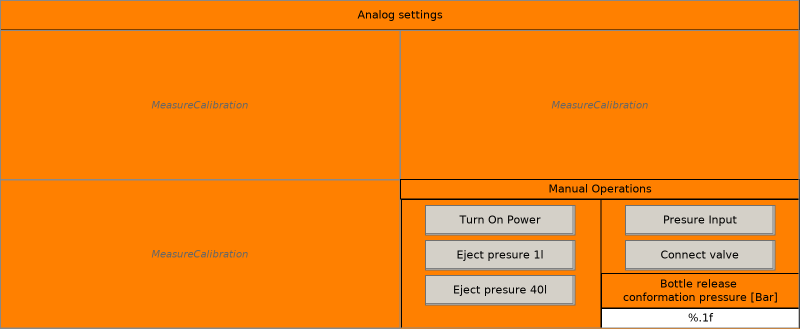
VISUALIZATION vService  // 800x329
VAR_IN_OUT
	fbChamber 	: fbChamber;
	stParams	: stParamsChamber;
END_VAR
    Rectangle (600,199 200x129)
    Rectangle (401,199 200x129)
    Rectangle (0,0 800x30), "Analog settings"
    Frame (0,30 400x150)
        shows MeasureCalibration(stMeasureData := stParams.stPressureSens, diAnalogIn := fbChamber.stInOuts.iPressureRaw, MeasureName := 'Presure Calibration')
    Frame (0,179 400x150)
        shows MeasureCalibration(stMeasureData := stParams.stVoltageSens, diAnalogIn := fbChamber.stInOuts.iVoltageRaw, MeasureName := 'Voltage Calibration')
    Frame (400,30 400x150)
        shows MeasureCalibration(stMeasureData := stParams.stCurrenteSens, diAnalogIn := fbChamber.stInOuts.iCurrentRaw, MeasureName := 'Curent Calibration')
    Rectangle (400,179 400x20), "Manual Operations"
    Button (425,205 150x30), "Turn On Power"
        OnMouseClick: toggle fbChamber.stInOuts.bPowerON
    Button (425,240 150x30), "Eject presure 1l"
        OnMouseClick: toggle fbChamber.stInOuts.bEjectPresure
    Button (425,275 150x30), "Eject presure 40l"
        OnMouseClick: toggle fbChamber.stInOuts.bEjectPresure40
    Button (625,205 150x30), "Presure Input"
        OnMouseClick: toggle fbChamber.stInOuts.bPressureIn
    Button (625,240 150x30), "Connect valve"
        OnMouseClick: toggle fbChamber.stInOuts.bBottle40l
    Rectangle (601,273 199x35), "Bottle release conformation pressure [Bar]"
    Rectangle (601,308 199x20), "%.1f", text variable: stParams.rMinimalPressure
        OnMouseClick: write the text variable via Default, min 0, max 1
END_VISUALIZATION

(* stored: Version 1.1.0.1, ProductVersion 3.1.4024.12
   Visu vService: Id {586c4eb4-97b8-461b-a26d-5fcf90b421b9} *)
